// TIA Portal project "WintonWasher_Recycler" (V15)

(* hardware
DEVICE "S7300/ET200M station_1"  S7-300 station
   slot 0: "Rail_0"  Rail  6ES7 390-1***0-0AA0
   slot 2: "PLC_1"  CPU 315-2 PN/DP  6ES7 315-2EH14-0AB0  V3.2
      slot 2: "PROFINET interface_1"  PN-IO
         slot 1: "Port_1"  Port
         slot 2: "Port_2"  Port
   slot 4: "DI 32x24VDC_1"  DI32 x 24VDC  6ES7 321-1BL00-0AA0
   slot 5: "DO 32x24VDC/0.5A_1"  DO32 x 24VDC / 0.5A  6ES7 322-1BL00-0AA0
DEVICE "HMI_1"  TP700 Comfort
   slot 0: "HMI_1"  TP700 Comfort  6AV2 124-0GC01-0AX0  15.0.0.0
   slot 1: "HMI_RT_1"  TP700 Comfort  6AV2 124-0GC01-0AX0  15.0.0.0
   slot 5: "HMI_1.IE_CP_1"  PROFINET Interface  15.0.0.0
      slot 1: "PROFINET Interface_1"  PROFINET Interface
         slot 1: "Port_1"  Port
         slot 2: "Port_2"  Port
   slot 7: "HMI_1.MPI/DP_CP_1"  MPI/DP Interface  15.0.0.0
DEVICE "GSD device_1"  GSD.Device
   slot 0: "Rack_0"  Rail
*)

// ===== PLC "PLC_1"  CPU 315-2 PN/DP =====

VAR_GLOBAL   // PLC tag table "Ouput Tag Table"
   "Qx Shear Cyl Ret" AT %Q10.0 : Bool;
   "Qx Shear Cyl Ext" AT %Q10.1 : Bool;   // lateral must be ret, punch must be ret
   "Qx Prestop Cyl Ret" AT %Q10.2 : Bool;   // RET lets part through
   "Qx Prestop Cyl Ext" AT %Q10.3 : Bool;
   "Qx Endstop Cyl Ret" AT %Q10.4 : Bool;   // prestop must be ext,
   "Qx Endstop Cyl Ext" AT %Q10.5 : Bool;
   "Qx Clamp Cyl Ret" AT %Q10.6 : Bool;
   "Qx Clamp Cyl Ext" AT %Q10.7 : Bool;
   "Qx Punch Cyl Ret" AT %Q11.0 : Bool;
   "Qx Punch Cyl Ext" AT %Q11.1 : Bool;
   "Qx Gripper Cyl Ret" AT %Q12.0 : Bool;
   "Qx Gripper Cyl Ext" AT %Q12.1 : Bool;
   "Qx Lat Cyl Ret" AT %Q12.2 : Bool;
   "Qx Lat Cyl Ext" AT %Q12.3 : Bool;   // Prestop must be EXT, gripper ret, endstop must be RET, punch ret, shear ret, clamps ret
   "Qx T2 Cyl Ret" AT %Q12.4 : Bool;
   "Qx T2 Cyl Ext" AT %Q12.5 : Bool;
   "Qx T1 Cyl Ret" AT %Q12.6 : Bool;
   "Qx T1 Cyl Ext" AT %Q12.7 : Bool;
   "Qx Cycle Start PL" AT %Q5.0 : Bool;
   "Qx Feeder OFF" AT %Q5.1 : Bool;   // Logic is Reversed!
   "Qx Overhead Light ON" AT %Q5.2 : Bool;
   "Qx Fan ON" AT %Q5.3 : Bool;
   "Qx Auxiliary Lights ON" AT %Q5.4 : Bool;
END_VAR

VAR_GLOBAL   // PLC tag table "Input Tag Table"
   "Ix Prestop Ext PX" AT %I10.2 : Bool;
   "Ix Prestop Ret PX" AT %I10.3 : Bool;
   "Ix Endstop Ext PX" AT %I10.4 : Bool;
   "Ix Endstop Ret PX" AT %I10.5 : Bool;
   "Ix Punch Ext PX" AT %I10.6 : Bool;
   "Ix Punch Ret PX" AT %I10.7 : Bool;
   "Ix Washer Present PX" AT %I11.0 : Bool;
   "Ix Left Clamp Ext PX" AT %I11.2 : Bool;
   "Ix Left Clamp Ret PX" AT %I11.3 : Bool;
   "Ix Right Clamp Ext PX" AT %I11.4 : Bool;
   "Ix Right Clamp Ret PX" AT %I11.5 : Bool;
   "Ix Left Shear Ext PX" AT %I11.6 : Bool;
   "Ix Left Shear Ret PX" AT %I11.7 : Bool;
   "Backup Washer Present PX" AT %I11.1 : Bool;
   "Ix Gripper Ext PX" AT %I12.0 : Bool;
   "Ix Gripper Ret PX" AT %I12.1 : Bool;
   "Ix Lat Ext PX" AT %I12.2 : Bool;
   "Ix Lat Ret PX" AT %I12.3 : Bool;
   "Ix T2 Ext PX" AT %I12.4 : Bool;
   "Ix T2 Ret PX" AT %I12.5 : Bool;
   "Ix T1 Ext PX" AT %I12.6 : Bool;
   "Ix T1 Ret PX" AT %I12.7 : Bool;
   "Ix Sense Part Ready PE" AT %I13.4 : Bool;
   "Ix Right Shear Ext PX" AT %I13.6 : Bool;
   "Ix Right Shear Ret PX" AT %I13.7 : Bool;
   "Ix Cycle Start PB" AT %I1.0 : Bool;
   "Ix ESTOP Not Pressed" AT %I1.1 : Bool;
   "Ix Doors Are Closed" AT %I1.2 : Bool;
END_VAR

DATA_BLOCK "DB_WintonWasher"   // DB1
{ S7_Optimized_Access := 'FALSE' }
VERSION : 0.1
// stored: InstanceOfName FB_WintonWasher
"FB_WintonWasher"
BEGIN
END_DATA_BLOCK

DATA_BLOCK "HMI_DB"   // DB7
{ S7_Optimized_Access := 'FALSE' }
VERSION : 0.1
   VAR
      MasterReset : Bool;
      Pause : Bool;
      "Auto On" : Bool;
      "Punch Ext" : Bool;
      "Punch Ret" : Bool;
      "Shear Ext" : Bool;
      "Shear Ret" : Bool;
      "Prestop Ext" : Bool;
      "Prestop Ret" : Bool;
      "Endstop Ext" : Bool;
      "Endstop Ret" : Bool;
      "Clamp Ext" : Bool;
      "Clamp Ret" : Bool;
      "Gripper Ext" : Bool;
      "Gripper Ret" : Bool;
      "Lat Ext" : Bool;
      "Lat Ret" : Bool;
      "T1 Ext" : Bool;
      "T1 Ret" : Bool;
      "T2 Ext" : Bool;
      "T2 Ret" : Bool;
      Vibrate : Bool;
      "Overhead Lights" : Bool;
      "Auxiliary Lights" : Bool;
      Fan : Bool;
      Bin_Count : Int;
      Reset_Bin_Count : Bool;
      Cycle_Count : Int;
   END_VAR
BEGIN
END_DATA_BLOCK

DATA_BLOCK "Alarms_DB"   // DB11
{ S7_Optimized_Access := 'FALSE' }
VERSION : 0.1
   VAR
      Alarms : Word;
   END_VAR
BEGIN
END_DATA_BLOCK

FUNCTION_BLOCK "FB_WintonWasher"   // FB1, STL
TITLE = Winton Washer Recycler
{ S7_Optimized_Access := 'FALSE' }
VERSION : 0.1
// Winton Washer Recycler Program
   VAR_INPUT
      "ESTOP Pressed" : Bool;
      "Ix Doors are Closed" : Bool;
      "Ix Prestop Ext PX" : Bool;
      "Ix Prestop Ret PX" : Bool;
      "Ix Endstop Ext PX" : Bool;
      "Ix Endstop Ret PX" : Bool;
      "Ix Punch Ext PX" : Bool;
      "Ix Punch Ret PX" : Bool;
      "Ix Washer Present PX" : Bool;
      "Ix Left Clamp Ext PX" : Bool;
      "Ix Left Clamp Ret PX" : Bool;
      "Ix Right Clamp Ext PX" : Bool;
      "Ix Right Clamp Ret PX" : Bool;
      "Ix Left Shear Ext PX" : Bool;
      "Ix Left Shear Ret PX" : Bool;
      "Backup Washer Present PX" : Bool;
      "Ix Gripper Ext PX" : Bool;
      "Ix Gripper Ret PX" : Bool;
      "Ix Lat Ext PX" : Bool;
      "Ix Lat Ret PX" : Bool;
      "Ix T2 Ext PX" : Bool;
      "Ix T2 Ret PX" : Bool;
      "Ix T1 Ext PX" : Bool;
      "Ix T1 Ret PX" : Bool;
      "Ix Sense Part Ready PE" : Bool;
      "Ix Right Shear Ext PX" : Bool;
      "Ix Right Shear Ret PX" : Bool;
      "Ix Cycle Start PB" : Bool;
   END_VAR
   VAR_OUTPUT
      "Qx Shear Cyl Ret" : Bool;
      "Qx Shear Cyl Ext" : Bool;
      "Qx Prestop Cyl Ret" : Bool;
      "Qx Prestop Cyl Ext" : Bool;
      "Qx Endstop Cyl Ret" : Bool;
      "Qx Endstop Cyl Ext" : Bool;
      "Qx Clamp Cyl Ret" : Bool;
      "Qx Clamp Cyl Ext" : Bool;
      "Qx Punch Cyl Ret" : Bool;
      "Qx Punch Cyl Ext" : Bool;
      "Qx Gripper Cyl Ret" : Bool;
      "Qx Gripper Cyl Ext" : Bool;
      "Qx Lat Cyl Ret" : Bool;
      "Qx Lat Cyl Ext" : Bool;
      "Qx T2 Cyl Ret" : Bool;
      "Qx T2 Cyl Ext" : Bool;
      "Qx T1 Cyl Ret" : Bool;
      "Qx T1 Cyl Ext" : Bool;
      "Qx Cycle Start PL" : Bool;
      "Qx Feeder OFF" : Bool;
      "Qx Overhead Light ON" : Bool;
      "Qx Fan ON" : Bool;
      "Qx Auxiliary Lights ON" : Bool;
   END_VAR
   VAR
      "Master Reset" : Bool;
      Pause : Bool;
      Auto : Struct
         "Shear Cyl Ret" : Bool;
         "Shear Cyl Ext" : Bool;
         "Prestop Cyl Ret" : Bool;
         "Prestop Cyl Ext" : Bool;
         "Endstop Cyl Ret" : Bool;
         "Endstop Cyl Ext" : Bool;
         "Clamp Cyl Ret" : Bool;
         "Clamp Cyl Ext" : Bool;
         "Punch Cyl Ret" : Bool;
         "Punch Cyl Ext" : Bool;
         "Gripper Cyl Ret" : Bool;
         "Gripper Cyl Ext" : Bool;
         "Lat Cyl Ret" : Bool;
         "Lat Cyl Ext" : Bool;
         "T2 Cyl Ret" : Bool;
         "T2 Cyl Ext" : Bool;
         "T1 Cyl Ret" : Bool;
         "T1 Cyl Ext" : Bool;
         "Cycle Start PL" : Bool;
         "Feeder OFF" : Bool;
      END_STRUCT;
      Manual : Struct
         "Shear Cyl Ret" : Bool;
         "Shear Cyl Ext" : Bool;
         "Prestop Cyl Ret" : Bool;
         "Prestop Cyl Ext" : Bool;
         "Endstop Cyl Ret" : Bool;
         "Endstop Cyl Ext" : Bool;
         "Clamp Cyl Ret" : Bool;
         "Clamp Cyl Ext" : Bool;
         "Punch Cyl Ret" : Bool;
         "Punch Cyl Ext" : Bool;
         "Gripper Cyl Ret" : Bool;
         "Gripper Cyl Ext" : Bool;
         "Lat Cyl Ret" : Bool;
         "Lat Cyl Ext" : Bool;
         "T2 Cyl Ret" : Bool;
         "T2 Cyl Ext" : Bool;
         "T1 Cyl Ret" : Bool;
         "T1 Cyl Ext" : Bool;
         "Cycle Start PL" : Bool;
         "Feeder OFF" : Bool;
         "Light ON" : Bool;
         "Fan ON" : Bool;
      END_STRUCT;
      "Step" : Struct
         Idle : Bool;
         "Sense Part Ready" : Bool;
         "Activate Prestop" : Bool;
         "Pick and Place Retract Endstop" : Bool;
         "Pick and Place Extend Lat Cyl" : Bool;
         "Pick and Place Extend Clamp" : Bool;
         "Pick and Place Extend Gripper" : Bool;
         "Pick and Place Retract Lat Cyl" : Bool;
         "Pick and Place Retract Gripper" : Bool;
         "Pick and Place Extend Endstop" : Bool;
         "Check for Washer" : Bool;
         "Open Path to Head Bin" : Bool;
         "Remove Head" : Bool;
         "Open Path to  Washer Bin" : Bool;
         "Retract Shears" : Bool;
         "Punch Out Washer" : Bool;
         "Retract Punch" : Bool;
         "Open Path to Body Bin" : Bool;
         "Drop Part" : Bool;
      END_STRUCT;
      Transition1_OK : Bool;
      Transition2_OK : Bool;
      Okay_toDelay1 : Bool;
      No_Parts_Error : Bool;
      "Enable PL Blink" : Bool;
      "Enable Overhead Blink" : Bool;
      Start_Delay_OffVibrate : Bool;
      Stop_Vibrate : Bool;   // timer output variable to stop feeder
      Washer_NotPresent : Bool;
      Bin_Overflow : Bool;
      Cyl_Jam : Bool;
      ClearPart : Struct
         "Retract Shears" : Bool;
         "Retract Punch" : Bool;
         "Extend Gripper" : Bool;
         "Retract Endstop" : Bool;
         "Extend Prestop" : Bool;
         "Retract Lateral" : Bool;
         "Retract Clamp" : Bool;
         "Reset Cyls for Idle" : Bool;
      END_STRUCT;
      "Start _Timeout" : Bool;
      Start_PreExt_Jam : Bool;
      Start_PreRet_Jam : Bool;
      Start_EndExt_Jam : Bool;
      Start_EndRet_Jam : Bool;
      Start_GrpExt_Jam : Bool;
      Start_GrpRet_Jam : Bool;
      Start_LatExt_Jam : Bool;
      Start_LatRet_Jam : Bool;
      Start_ShrExt_Jam : Bool;
      Start_ShrRet_Jam : Bool;
      Start_PunExt_Jam : Bool;
      Start_PunRet_Jam : Bool;
      Start_T1Ext_Jam : Bool;
      Start_T1Ret_Jam : Bool;
      Start_T2Ext_Jam : Bool;
      Start_T2Ret_Jam : Bool;
      Start_ClmpExt_Jam : Bool;
      Start_ClmpRet_Jam : Bool;
   END_VAR
BEGIN

REGION Network 1: Reset and Pause
   // Reset Conditions
   // Resets current machine state to Idle
   // HMI 'MASTER RESET' for cylinder fault or jam. 
   // -This button will automatically clear a part and reset cylinder positions to where they should be in Idle.
   ////////////////////////////////////////////////////
   //--------------Master Reset Conditions-------------
         A     #"ESTOP Pressed";
         =     #"Master Reset";

   ////////////////////////////////////////////////////
   //--------------Reset State Condition-------------
   //add other errors
         A     #"Master Reset";
         O     #No_Parts_Error;
         O(;
   //logic from "Clear part" sequence
         A     #ClearPart."Reset Cyls for Idle";
         A     #"Ix Gripper Ret PX";
         A     #"Ix Endstop Ext PX";
         A     #"Ix T1 Ret PX";
         A     #"Ix T2 Ext PX";
         );
         S     #"Step".Idle;
         R     #"Step"."Activate Prestop";
         R     #"Step"."Check for Washer";
         R     #"Step"."Drop Part";
         R     #"Step"."Open Path to  Washer Bin";
         R     #"Step"."Open Path to Body Bin";
         R     #"Step"."Open Path to Head Bin";
         R     #"Step"."Pick and Place Retract Endstop";
         R     #"Step"."Pick and Place Extend Lat Cyl";
         R     #"Step"."Pick and Place Extend Clamp";
         R     #"Step"."Pick and Place Extend Gripper";
         R     #"Step"."Pick and Place Retract Lat Cyl";
         R     #"Step"."Pick and Place Retract Gripper";
         R     #"Step"."Pick and Place Extend Endstop";
         R     #"Step"."Punch Out Washer";
         R     #"Step"."Remove Head";
         R     #"Step"."Retract Shears";
         R     #"Step"."Sense Part Ready";
         R     #ClearPart."Extend Gripper";
         R     #ClearPart."Extend Prestop";
         R     #ClearPart."Reset Cyls for Idle";
         R     #ClearPart."Retract Clamp";
         R     #ClearPart."Retract Endstop";
         R     #ClearPart."Retract Lateral";
         R     #ClearPart."Retract Punch";
         R     #ClearPart."Retract Shears";



   //////////////////////////////////////////////////////
   //--------------HMI Master Reset Response-------------
   //start clear part sequence
         A     "HMI_DB".MasterReset;
         S     #ClearPart."Retract Shears";
         R     #"Step"."Activate Prestop";
         R     #"Step"."Check for Washer";
         R     #"Step"."Drop Part";
         R     #"Step"."Open Path to  Washer Bin";
         R     #"Step"."Open Path to Body Bin";
         R     #"Step"."Open Path to Head Bin";
         R     #"Step"."Pick and Place Retract Endstop";
         R     #"Step"."Pick and Place Extend Lat Cyl";
         R     #"Step"."Pick and Place Extend Clamp";
         R     #"Step"."Pick and Place Extend Gripper";
         R     #"Step"."Pick and Place Retract Lat Cyl";
         R     #"Step"."Pick and Place Retract Gripper";
         R     #"Step"."Pick and Place Extend Endstop";
         R     #"Step"."Punch Out Washer";
         R     #"Step"."Remove Head";
         R     #"Step"."Retract Shears";
         R     #"Step"."Sense Part Ready";
         R     #"Step".Idle;

   ////////////////////////////////////////////
   //--------------Pause Logic-----------------
         AN    #"Ix Doors are Closed";
   // ON    "HMI_DB"."Auto On"
         O     "HMI_DB".Pause;
         =     #Pause;

   //use this timer to generate any delay desired
   //CALL  TON , "CylJam_Timer"
   //         time_type:=Time
   //         IN :=#Step."Retract Shears"
   //         PT :=T#2s
   //         Q  :=#Auto."Shear Cyl Ret"
   //         ET :=
END_REGION

REGION Network 2: Manual Network
   // Manual Control of all Outputs via HMI
   ////////////////////////////////////////////
   //--------------Manual: Prestop-------------
         A     "HMI_DB"."Prestop Ext";
         AN    "HMI_DB"."Auto On";
         =     #Manual."Prestop Cyl Ext";

         A     "HMI_DB"."Prestop Ret";
         AN    "HMI_DB"."Auto On";
         =     #Manual."Prestop Cyl Ret";

   ////////////////////////////////////////////
   //--------------Manual: Endsotp-------------
         A     "HMI_DB"."Endstop Ext";
         AN    "HMI_DB"."Auto On";
         =     #Manual."Endstop Cyl Ext";

         A     "HMI_DB"."Endstop Ret";
         AN    "HMI_DB"."Auto On";
         =     #Manual."Endstop Cyl Ret";

   ////////////////////////////////////////////
   //--------------Manual: Lateral-------------
         A     "HMI_DB"."Lat Ext";
         AN    "HMI_DB"."Auto On";
         =     #Manual."Lat Cyl Ext";

         A     "HMI_DB"."Lat Ret";
         AN    "HMI_DB"."Auto On";
         =     #Manual."Lat Cyl Ret";

   ////////////////////////////////////////////
   //--------------Manual: Gripper-------------
         A     "HMI_DB"."Gripper Ext";
         AN    "HMI_DB"."Auto On";
         =     #Manual."Gripper Cyl Ext";

         A     "HMI_DB"."Gripper Ret";
         AN    "HMI_DB"."Auto On";
         =     #Manual."Gripper Cyl Ret";

   ////////////////////////////////////////////
   //--------------Manual: Shears-------------
         A     "HMI_DB"."Shear Ext";
         AN    "HMI_DB"."Auto On";
         =     #Manual."Shear Cyl Ext";

         A     "HMI_DB"."Shear Ret";
         AN    "HMI_DB"."Auto On";
         =     #Manual."Shear Cyl Ret";

   ////////////////////////////////////////////
   //--------------Manual: Clamps-------------
         A     "HMI_DB"."Clamp Ext";
         AN    "HMI_DB"."Auto On";
         =     #Manual."Clamp Cyl Ext";

         A     "HMI_DB"."Clamp Ret";
         AN    "HMI_DB"."Auto On";
         =     #Manual."Clamp Cyl Ret";

   ////////////////////////////////////////////
   //--------------Manual: Washer Punch-------------
         A     "HMI_DB"."Punch Ext";
         AN    "HMI_DB"."Auto On";
         =     #Manual."Punch Cyl Ext";

         A     "HMI_DB"."Punch Ret";
         AN    "HMI_DB"."Auto On";
         =     #Manual."Punch Cyl Ret";

   ////////////////////////////////////////////
   //--------------Manual: Trap Door 1-------------
         A     "HMI_DB"."T1 Ext";
         AN    "HMI_DB"."Auto On";
         =     #Manual."T1 Cyl Ext";

         A     "HMI_DB"."T1 Ret";
         AN    "HMI_DB"."Auto On";
         =     #Manual."T1 Cyl Ret";


   ////////////////////////////////////////////
   //--------------Manual: Trap Door 2-------------
         A     "HMI_DB"."T2 Ext";
         AN    "HMI_DB"."Auto On";
         =     #Manual."T2 Cyl Ext";

         A     "HMI_DB"."T2 Ret";
         AN    "HMI_DB"."Auto On";
         =     #Manual."T2 Cyl Ret";

   ////////////////////////////////////////////
   //--------------Manual: Vibrate Feeder-------------
         AN    "HMI_DB".Vibrate;
         AN    "HMI_DB"."Auto On";
         =     #Manual."Feeder OFF";
END_REGION

REGION Network 3: Auto Sequence - Step Transitions
   // How the auto sequence transitions states
   ////////////////////////////////////////////////////
   //-------------Idle to Sense Part Ready-------------
         A     #"Step".Idle;
         R     #ClearPart."Reset Cyls for Idle";

         A     #"Step".Idle;
         A     #"Ix Cycle Start PB";
         A     "HMI_DB"."Auto On";
         AN    #Pause;
         AN    "Bin_Count".Q;
         R     #"Step".Idle;
         S     #"Step"."Sense Part Ready";


   ////////////////////////////////////////////////////
   //--------sense part ready to activate prestop------
         A     #"Step"."Sense Part Ready";
         A     #"Ix Sense Part Ready PE";
         A     "HMI_DB"."Auto On";
         AN    #Pause;
         S     #"Step"."Activate Prestop";
         R     #"Step"."Sense Part Ready";

         A     #"Step"."Sense Part Ready";
         AN    "Bin_Count".Q;
         =     #"Start _Timeout";

   //No parts timeout delay
         CALL  TON , "No Parts Timeout Timer"
         ( IN := #"Start _Timeout",
           PT := T#30s,
           Q  := #No_Parts_Error,
           ET :=
         );

   ////////////////////////////////////////////////////
   //-------Activate prestop to Pick and Place---------
         A     #"Step"."Activate Prestop";
         A     #"Ix Prestop Ext PX";
         A     "HMI_DB"."Auto On";
         AN    #Pause;
         S     #"Step"."Pick and Place Retract Endstop";
         R     #"Step"."Activate Prestop";

   ////////////////////////////////////////////////////
   //---------------Pick and place---------------------
   //---------------retract endstop--------------------
         A     #"Step"."Pick and Place Retract Endstop";
         A     #"Ix Endstop Ret PX";
         A     "HMI_DB"."Auto On";
         AN    #Pause;
         R     #"Step"."Pick and Place Retract Endstop";
         S     #"Step"."Pick and Place Extend Lat Cyl";

   ////////////////////////////////////////////////////
   //---------------Pick and place---------------------
   //---------------Extend Lateral---------------------
         A     #"Step"."Pick and Place Extend Lat Cyl";
         A     #"Ix Lat Ext PX";
         A     "HMI_DB"."Auto On";
         AN    #Pause;
         R     #"Step"."Pick and Place Extend Lat Cyl";
         S     #"Step"."Pick and Place Extend Clamp";

   ////////////////////////////////////////////////////
   //---------------Pick and place---------------------
   //---------------Extend Clamp-----------------------
         A     #"Step"."Pick and Place Extend Clamp";
         A     #"Ix Left Clamp Ext PX";
         A     #"Ix Right Clamp Ext PX";
         A     "HMI_DB"."Auto On";
         AN    #Pause;
         R     #"Step"."Pick and Place Extend Clamp";
         S     #"Step"."Pick and Place Extend Gripper";

   ////////////////////////////////////////////////////
   //---------------Pick and place---------------------
   //---------------Extend Gripper---------------------
         A     #"Step"."Pick and Place Extend Gripper";
         A     #"Ix Gripper Ext PX";
         A     "HMI_DB"."Auto On";
         AN    #Pause;
         R     #"Step"."Pick and Place Extend Gripper";
         S     #"Step"."Pick and Place Retract Lat Cyl";

   ////////////////////////////////////////////////////
   //---------------Pick and place---------------------
   //---------------Retract Lateral--------------------
         A     #"Step"."Pick and Place Retract Lat Cyl";
         A     #"Ix Lat Ret PX";
         A     "HMI_DB"."Auto On";
         AN    #Pause;
         R     #"Step"."Pick and Place Retract Lat Cyl";
         S     #"Step"."Pick and Place Retract Gripper";

   ////////////////////////////////////////////////////
   //---------------Pick and place---------------------
   //---------------Retract Gripper--------------------
         A     #"Step"."Pick and Place Retract Gripper";
         A     #"Ix Gripper Ret PX";
         A     "HMI_DB"."Auto On";
         AN    #Pause;
         R     #"Step"."Pick and Place Retract Gripper";
         S     #"Step"."Pick and Place Extend Endstop";

   ////////////////////////////////////////////////////
   //---------------Pick and place---------------------
   //---------------Extend Endstop--------------------
         A     #"Step"."Pick and Place Extend Endstop";
         A     #"Ix Endstop Ext PX";
         A     "HMI_DB"."Auto On";
         AN    #Pause;
         R     #"Step"."Pick and Place Extend Endstop";
         S     #"Step"."Check for Washer";

   ////////////////////////////////////////////////////
   //----check for washer to Open Path to Head Bin-----
         A     #"Step"."Check for Washer";
         A     #"Ix Washer Present PX";
         A     "HMI_DB"."Auto On";
         AN    #Pause;
         R     #"Step"."Check for Washer";
         S     #"Step"."Open Path to Head Bin";

   //else
   //timer, put output of timer on Drop part conditions

   ////////////////////////////////////////////////////
   //---------check for washer to Drop part, put in condition for drp part
         CALL  TON , "Washer Not Present Timeout Timer"
         ( IN := #"Step"."Check for Washer",
           PT := T#100ms,
           Q  := #Washer_NotPresent,
           ET :=
         );

   //      A     #Step."Check for Washer"
   //      A   Check for Washer Timeout
   //      S     #Step."Drop Part"
   //      R     #Step."Check for Washer"

   ////////////////////////////////////////////////////
   //---------Open Path to Head Bin, to Remove Head---
         A     #"Step"."Open Path to Head Bin";
         A     #"Ix T1 Ext PX";
         A     #"Ix T2 Ext PX";
         A     "HMI_DB"."Auto On";
         AN    #Pause;
         S     #"Step"."Remove Head";
         R     #"Step"."Open Path to Head Bin";

   ////////////////////////////////////////////////////
   //------Remove Head, to Open Path to Washer Bin-----
   //start delay after Extension
         A     #"Step"."Remove Head";
         A     #"Ix Left Shear Ext PX";
         =     #Okay_toDelay1;

   //delay
         CALL  TON , "Delay_Transition_toWasherBin"
         ( IN := #Okay_toDelay1,
           PT := T#1s,
           Q  := #Transition1_OK,
           ET :=
         );

         A     #"Step"."Remove Head";
         A     #"Ix Left Shear Ext PX";
         A     #"Ix Right Shear Ext PX";
         A     #Transition1_OK;
         A     "HMI_DB"."Auto On";
         AN    #Pause;
         R     #"Step"."Remove Head";
         S     #"Step"."Open Path to  Washer Bin";

   ////////////////////////////////////////////////////
   //-----Open Path to Washer Bin to Retract Shears----
         A     #"Step"."Open Path to  Washer Bin";
         A     #"Ix T1 Ext PX";
         A     #"Ix T2 Ret PX";
         A     "HMI_DB"."Auto On";
         AN    #Pause;
         R     #"Step"."Open Path to  Washer Bin";
         S     #"Step"."Retract Shears";

   ////////////////////////////////////////////////////
   //---------Retract Shears to Punch Out Washer-------
         A     #"Step"."Retract Shears";
         A     #"Ix Left Shear Ret PX";
         A     #"Ix Right Shear Ret PX";
         A     "HMI_DB"."Auto On";
         AN    #Pause;
         R     #"Step"."Retract Shears";
         S     #"Step"."Punch Out Washer";


   ////////////////////////////////////////////////////
   //-----Punch Out Washer to Retract Punch----
         A     #"Step"."Punch Out Washer";
         A     #"Ix Punch Ext PX";
         A     "HMI_DB"."Auto On";
         AN    #Pause;
         R     #"Step"."Punch Out Washer";
         S     #"Step"."Retract Punch";

   ////////////////////////////////////////////////////
   //-----Retract Punch to Open Path to Body Bin-------
   //delay
         CALL  TON , "Delay_Transition_toBodyBin"
         ( IN := #"Step"."Retract Punch",
           PT := T#1s,
           Q  := #Transition2_OK,
           ET :=
         );

         A     #"Step"."Retract Punch";
         A     #"Ix Punch Ret PX";
         A     "HMI_DB"."Auto On";
         AN    #Pause;
         A     #Transition2_OK;
         R     #"Step"."Retract Punch";
         S     #"Step"."Open Path to Body Bin";

   ////////////////////////////////////////////////////
   //-------Open Pach to Body Bin to Drop Part---------
         A(;
         A     #"Step"."Open Path to Body Bin";
         A     #"Ix T1 Ret PX";
         );
         O(;
         A     #"Step"."Check for Washer";
         A     #Washer_NotPresent;
         );
         A     "HMI_DB"."Auto On";
         AN    #Pause;
         R     #"Step"."Open Path to Body Bin";
         R     #"Step"."Check for Washer";
         S     #"Step"."Drop Part";

   ////////////////////////////////////////////////////
   //---------Drop Part to Wait for Part Ready---------
         A     #"Step"."Drop Part";
         A     #"Ix Left Clamp Ret PX";
         A     #"Ix Right Clamp Ret PX";
         A     "HMI_DB"."Auto On";
         AN    #Pause;
         R     #"Step"."Drop Part";
         S     #"Step"."Sense Part Ready";
END_REGION

REGION Network 4: Auto Sequence - Outputs
   ////////////////////////////////////////////////////////////////////////
   //--------------------------Idle----------------------------------------

   //cycle start PL
         A     #"Step".Idle;
         A     "HMI_DB"."Auto On";
         AN    "PL_Blink".Q;
         =     #"Enable PL Blink";

         CALL  TON , "PL_Blink"
         ( IN := #"Enable PL Blink",
           PT := T#1s,
           Q  := ,
           ET :=
         );


         AN    #"Step".Idle;
         AN    #Pause;
         A     "HMI_DB"."Auto On";
         AN    "HMI_DB".MasterReset;
         O(;
         L     "PL_Blink".ET;
         L     T#500ms;
         >D;
         );
         =     #Auto."Cycle Start PL";

   ////////////////////////////////////////////////////////////////////////
   //--------------------------Sense Part Ready----------------------------
   //     A     #"Ix Sense Part Ready PE"
   //   AN    "Bin_Count".Q
   //  =     #Start_Delay_OffVibrate

   //Vibrating Feeder control (inversed)
   //delay after seeing part to remove time inbetween cycles
         CALL  TOF , "Delay_VibrateOFF"
         ( IN := #"Ix Sense Part Ready PE",
           PT := T#2s,
           Q  := #Stop_Vibrate,
           ET :=
         );

   //if neither are true, it is OFF
         AN    #"Step"."Sense Part Ready";
         AN    #Stop_Vibrate;
         ON    "HMI_DB"."Auto On";
         O     #"Master Reset";
         O     "Bin_Count".Q;
         =     #Auto."Feeder OFF";

   //retract prestop
         A     #"Step"."Sense Part Ready";
         =     #Auto."Prestop Cyl Ret";

   ////////////////////////////////////////////////////////////////////////
   //--------------------------Activate Prestop----------------------------
   //Extend Prestop
         A     #"Step"."Activate Prestop";
         =     #Auto."Prestop Cyl Ext";

   ////////////////////////////////////////////////////////////////////////
   //-----------------Pick and Place Retract Endstop-----------------------
   //retract endstop
         A     #"Step"."Pick and Place Retract Endstop";
         =     #Auto."Endstop Cyl Ret";

   ////////////////////////////////////////////////////////////////////////
   //-----------------Pick and Place Extend Lat Cyl-----------------------
   //retract endstop
         A     #"Step"."Pick and Place Extend Lat Cyl";
         =     #Auto."Lat Cyl Ext";

   ////////////////////////////////////////////////////////////////////////
   //-----------------Pick and Place Extend Clamp-----------------------
         A     #"Step"."Pick and Place Extend Clamp";
         =     #Auto."Clamp Cyl Ext";

   ////////////////////////////////////////////////////////////////////////
   //-----------------Pick and Place Extend Gripper-----------------------
         A     #"Step"."Pick and Place Extend Gripper";
         =     #Auto."Gripper Cyl Ext";

   ////////////////////////////////////////////////////////////////////////
   //-----------------Pick and Place Retract Lateral-----------------------
         A     #"Step"."Pick and Place Retract Lat Cyl";
         =     #Auto."Lat Cyl Ret";

   ////////////////////////////////////////////////////////////////////////
   //-----------------Pick and Place Retract Gripper-----------------------
         A     #"Step"."Pick and Place Retract Gripper";
         =     #Auto."Gripper Cyl Ret";

   ////////////////////////////////////////////////////////////////////////
   //-----------------Pick and Place Extend Endstop-----------------------
         A     #"Step"."Pick and Place Extend Endstop";
         =     #Auto."Endstop Cyl Ext";

   ////////////////////////////////////////////////////////////////////////
   //-------------------------Check for Washer-----------------------------

   ////////////////////////////////////////////////////////////////////////
   //-----------------------Open Path(s) logic--------------------------

   //T1
         A     #"Step"."Open Path to Head Bin";
         O     #"Step"."Open Path to  Washer Bin";
         =     #Auto."T1 Cyl Ext";

   //T2
         A     #"Step"."Open Path to Head Bin";
         O     #"Step"."Open Path to Body Bin";
         =     #Auto."T2 Cyl Ext";


   //T1
         A     #"Step"."Open Path to Body Bin";
         =     #Auto."T1 Cyl Ret";

   //T2
         A     #"Step"."Open Path to  Washer Bin";
         =     #Auto."T2 Cyl Ret";

   ////////////////////////////////////////////////////////////////////////
   //---------------------------Remove Head--------------------------------
         A     #"Step"."Remove Head";
         =     #Auto."Shear Cyl Ext";

   ////////////////////////////////////////////////////////////////////////
   //-------------------------Open Path to Washer Bin-----------------------------
   //this logic is with the T1 and T2 logic

   ////////////////////////////////////////////////////////////////////////
   //-------------------------Retract Shears-----------------------------
         A     #"Step"."Retract Shears";
         =     #Auto."Shear Cyl Ret";

   ////////////////////////////////////////////////////////////////////////
   //-------------------------Punch Out Washer-----------------------------
         A     #"Step"."Punch Out Washer";
         =     #Auto."Punch Cyl Ext";

   ////////////////////////////////////////////////////////////////////////
   //-------------------------Retract Punch-----------------------------
         A     #"Step"."Retract Punch";
         =     #Auto."Punch Cyl Ret";


   ////////////////////////////////////////////////////////////////////////
   //-------------------------Drop Part-----------------------------
         A     #"Step"."Drop Part";
         =     #Auto."Clamp Cyl Ret";

         CALL  CTU, "Bin_Count"
         ( CU := #"Step"."Drop Part",
           R  := "HMI_DB".Reset_Bin_Count,
           PV := 135,
           Q  := #Bin_Overflow,
           CV := "HMI_DB".Bin_Count
         );

         CALL  CTU , "Cycle_Count"
         ( CU := #"Step"."Drop Part",
           R  := ,
           PV := 32767,
           Q  := ,
           CV := "HMI_DB".Cycle_Count
         );


   //and increment a monthly cycle count
END_REGION

REGION Network 5: Outputs
   // Output Buffering
   ////////////////////////////////////////////////////////////////////////
   //-----------------------PLC Output Card--------------------------------

   //feeder
         A     #Auto."Feeder OFF";
         O(;
         A     #"Step".Idle;
         A     #Manual."Feeder OFF";
         AN    "HMI_DB"."Auto On";
         );
         O     #Cyl_Jam;
         O     #"Master Reset";
         =     #"Qx Feeder OFF";

   //overhead light, manually controlled
         A     "HMI_DB"."Overhead Lights";
         AN    #Cyl_Jam;
         O(;
         L     "Overhead_Blink".ET;
         L     T#500ms;
         >D;
         );
         =     #"Qx Overhead Light ON";

   //Aux Lights, manually controlled
         A     "HMI_DB"."Auxiliary Lights";
         =     #"Qx Auxiliary Lights ON";

   //Fan, manually controlled
         A     "HMI_DB".Fan;
         =     #"Qx Fan ON";

   //cycle start pilot light
         A     #Auto."Cycle Start PL";
         =     #"Qx Cycle Start PL";

   ////////////////////////////////////////////////////////////////////////
   //-----------------------Output Bank Cyls--------------------------------
   //////////////-----Contains interlocking cyl conditions-------///////////
   ////prestop
         A     #Auto."Prestop Cyl Ext";
         O     #ClearPart."Extend Prestop";
         O     #Manual."Prestop Cyl Ext";
         AN    #"Ix Prestop Ext PX";
         AN    #Cyl_Jam;
         =     #"Qx Prestop Cyl Ext";

         A     #Auto."Prestop Cyl Ret";
         O     #Manual."Prestop Cyl Ret";
         AN    #"Ix Prestop Ret PX";
         AN    #Cyl_Jam;
         =     #"Qx Prestop Cyl Ret";

   ////endstop
         A     #Auto."Endstop Cyl Ext";
         O     #ClearPart."Reset Cyls for Idle";
         O     #Manual."Endstop Cyl Ext";
         AN    #"Ix Endstop Ext PX";
         AN    #Cyl_Jam;
         =     #"Qx Endstop Cyl Ext";

         A     #Auto."Endstop Cyl Ret";
         O     #ClearPart."Retract Endstop";
         O     #Manual."Endstop Cyl Ret";
         AN    #"Ix Endstop Ret PX";
         AN    #Cyl_Jam;
         =     #"Qx Endstop Cyl Ret";

   ////gripper
         A     #Auto."Gripper Cyl Ext";
         O     #ClearPart."Extend Gripper";
         O     #Manual."Gripper Cyl Ext";
         AN    #"Ix Gripper Ext PX";
         AN    #Cyl_Jam;
         =     #"Qx Gripper Cyl Ext";

         A     #Auto."Gripper Cyl Ret";
         O     #ClearPart."Reset Cyls for Idle";
         O     #Manual."Gripper Cyl Ret";
         AN    #"Ix Gripper Ret PX";
         AN    #Cyl_Jam;
         =     #"Qx Gripper Cyl Ret";

   ////lateral cyl
         A     #Auto."Lat Cyl Ext";
         O     #Manual."Lat Cyl Ext";
         A     #"Ix Prestop Ext PX";
         A     #"Ix Endstop Ret PX";
         A     #"Ix Punch Ret PX";
         A     #"Ix Left Shear Ret PX";
         A     #"Ix Right Shear Ret PX";
         A     #"Ix Left Clamp Ret PX";
         A     #"Ix Right Clamp Ret PX";
         AN    #"Ix Lat Ext PX";
         AN    #Cyl_Jam;
         =     #"Qx Lat Cyl Ext";

         A     #Auto."Lat Cyl Ret";
         O     #ClearPart."Retract Lateral";
         O     #Manual."Lat Cyl Ret";
         A     #"Ix Prestop Ext PX";
         A     #"Ix Endstop Ret PX";
         A     #"Ix Punch Ret PX";
         A     #"Ix Left Shear Ret PX";
         A     #"Ix Right Shear Ret PX";
         AN    #"Ix Lat Ret PX";
         AN    #Cyl_Jam;
         =     #"Qx Lat Cyl Ret";

   //clamp cyl
         A     #Auto."Clamp Cyl Ret";
         O     #ClearPart."Retract Clamp";
         O     #Manual."Clamp Cyl Ret";
         A(;
         ON    #"Ix Left Clamp Ret PX";
         ON    #"Ix Right Clamp Ret PX";
         );
         AN    #Cyl_Jam;
         =     #"Qx Clamp Cyl Ret";

         A(;
         A     #Auto."Clamp Cyl Ext";
         O     #Manual."Clamp Cyl Ext";
         A(;
         ON    #"Ix Left Clamp Ext PX";
         ON    #"Ix Right Clamp Ext PX";
         );
         );
   //these ensure part is clamped while sheared and punched
         O     #"Step"."Remove Head";
         AN    #Okay_toDelay1;
         O     #"Step"."Punch Out Washer";
         AN    #Cyl_Jam;
         =     #"Qx Clamp Cyl Ext";

   //T1 Cyl
         A     #Auto."T1 Cyl Ext";
         O     #Manual."T1 Cyl Ext";
         AN    #"Ix T1 Ext PX";
         AN    #Cyl_Jam;
         =     #"Qx T1 Cyl Ext";

         A     #Auto."T1 Cyl Ret";
         O     #ClearPart."Retract Shears";
         O     #Manual."T1 Cyl Ret";
         AN    #"Ix T1 Ret PX";
         AN    #Cyl_Jam;
         =     #"Qx T1 Cyl Ret";

   //T2 cyl
         A     #Auto."T2 Cyl Ext";
         O     #Manual."T2 Cyl Ext";
         O     #ClearPart."Reset Cyls for Idle";
         AN    #"Ix T2 Ext PX";
         AN    #Cyl_Jam;
         =     #"Qx T2 Cyl Ext";

         A     #Auto."T2 Cyl Ret";
         O     #Manual."T2 Cyl Ret";
         AN    #"Ix T2 Ret PX";
         AN    #Cyl_Jam;
         =     #"Qx T2 Cyl Ret";

   //shear cyl
         A     #Auto."Shear Cyl Ext";
         O     #Manual."Shear Cyl Ext";
         A     #"Ix Lat Ret PX";
         A     #"Ix Punch Ret PX";
         A(;
         ON    #"Ix Left Shear Ext PX";
         ON    #"Ix Right Shear Ext PX";
         );
         AN    #Cyl_Jam;
         =     #"Qx Shear Cyl Ext";

         A     #Auto."Shear Cyl Ret";
         O     #ClearPart."Retract Shears";
         O     #Manual."Shear Cyl Ret";
         A(;
         ON    #"Ix Left Shear Ret PX";
         ON    #"Ix Right Shear Ret PX";
         );
         AN    #Cyl_Jam;
         =     #"Qx Shear Cyl Ret";

   //punch cyl
         A     #Auto."Punch Cyl Ext";
         O     #Manual."Punch Cyl Ext";
         A     #"Ix Left Shear Ret PX";
         A     #"Ix Right Shear Ret PX";
         AN    #"Ix Punch Ext PX";
         AN    #Cyl_Jam;
         =     #"Qx Punch Cyl Ext";

         A     #Auto."Punch Cyl Ret";
         O     #ClearPart."Retract Punch";
         O     #Manual."Punch Cyl Ret";
         A     #"Ix Left Shear Ret PX";
         A     #"Ix Right Shear Ret PX";
         AN    #"Ix Punch Ret PX";
         AN    #Cyl_Jam;
         =     #"Qx Punch Cyl Ret";
END_REGION

REGION Network 6: Clear Part
   // Clears Part or Jam (potentially) from loading process. 
   // Pressing "MASTER RESET" on HMI triggers this sequence. 
   // Goes to idle when complete
   //state logic
   ////////////////////////////////////////////////////
   //---------Retract Shears to Retract Punch-------
         A     #ClearPart."Retract Shears";
         A     #"Ix Left Shear Ret PX";
         A     #"Ix Right Shear Ret PX";
         A     #"Ix T1 Ret PX";
         AN    #Pause;
         R     #ClearPart."Retract Shears";
         S     #ClearPart."Retract Punch";

   ////////////////////////////////////////////////////
   //---------Retract Punch to Extend Gripper-------
         A     #ClearPart."Retract Punch";
         A     #"Ix Punch Ret PX";
         AN    #Pause;
         R     #ClearPart."Retract Punch";
         S     #ClearPart."Extend Gripper";

   ////////////////////////////////////////////////////
   //---------Extend Gripper to Retract Endstop-------
         A(;
         A     #ClearPart."Extend Gripper";
         A     #"Ix Gripper Ext PX";
         );
         O(;
         A     #ClearPart."Extend Gripper";
         A     #"Ix Lat Ret PX";
         );
         AN    #Pause;
         R     #ClearPart."Extend Gripper";
         S     #ClearPart."Retract Endstop";

   ////////////////////////////////////////////////////
   //---------Retract Endstop to Extend Prestop-------
         A(;
         A     #ClearPart."Retract Endstop";
         A     #"Ix Endstop Ret PX";
         );
         O(;
         A     #ClearPart."Retract Endstop";
         A     #"Ix Lat Ret PX";
         );
         AN    #Pause;
         R     #ClearPart."Retract Endstop";
         S     #ClearPart."Extend Prestop";

   ////////////////////////////////////////////////////
   //---------Extend Prestop to Retract Lateral-------
         A     #ClearPart."Extend Prestop";
         A     #"Ix Prestop Ext PX";
         AN    #Pause;
         R     #ClearPart."Extend Prestop";
         S     #ClearPart."Retract Lateral";

   ////////////////////////////////////////////////////
   //---------Retract Lateral to Retract Clamp-------
         A     #ClearPart."Retract Lateral";
         A     #"Ix Lat Ret PX";
         AN    #Pause;
         R     #ClearPart."Retract Lateral";
         S     #ClearPart."Retract Clamp";

   ////////////////////////////////////////////////////
   //---------Retract Clamp to Reset Cyls For Idle-------
         A     #ClearPart."Retract Clamp";
         A     #"Ix Left Clamp Ret PX";
         A     #"Ix Right Clamp Ret PX";
         AN    #Pause;
         R     #ClearPart."Retract Clamp";
         S     #ClearPart."Reset Cyls for Idle";

   ///////////////////////////////////////////////
   //reset other cyls
   //this logic is actually in "Idle" logic because it must be in the same 'rung'
   //   A     #ClearPart."Reset Cyls for Idle"
   //   A     #"Ix Gripper Ret PX"
   //   A     #"Ix Endstop Ext PX"
   //   A     #"Ix T1 Ret PX"
   //   A     #"Ix T2 Ext PX"
   //  R     #ClearPart."Reset Cyls for Idle"
   /////////////////  S     #Step.Idle

   ////////////////////////////////////////////////////////////////////////
   //end
END_REGION

REGION Network 7: Alarms
   // Because the HMI Alarms only works with INT data type, must set the individual address of the Data Block created: Alarms_DB
   //ESTOP
         A     #"ESTOP Pressed";
         =     %DB11.DBX0.0;

   //Doors
         AN    #"Ix Doors are Closed";
         =     %DB11.DBX0.1;

   //No Parts Timeout
         A     #No_Parts_Error;
         S     %DB11.DBX0.2;

   //bin is full
         A     "Bin_Count".Q;
         =     %DB11.DBX0.3;
END_REGION

REGION Network 8: Cylinder Jams
   // Cylinder Jam Logic for each ext and retract signal. 
   // Each one is 2 seconds and can be adjusted
   //blink Overhead lights when jammed
         A     #Cyl_Jam;
         AN    "Overhead_Blink".Q;
         =     #"Enable Overhead Blink";

         CALL  TON , "Overhead_Blink"
         ( IN := #"Enable Overhead Blink",
           PT := T#1s,
           Q  := ,
           ET :=
         );


   //------------------------------------------------------------
   //prestop
         A     #Auto."Prestop Cyl Ext";
         O     #Manual."Prestop Cyl Ext";
         O     #ClearPart."Extend Prestop";
         AN    #"Ix Prestop Ext PX";
         AN    #Pause;
         =     #Start_PreExt_Jam;

         CALL  TON, "Prestop_Ext_Jam_timer"
         ( IN := #Start_PreExt_Jam,
           PT := T#2s,
           Q  := ,
           ET :=
         );


         A     #Auto."Prestop Cyl Ret";
         O     #Manual."Prestop Cyl Ret";
         AN    #"Ix Prestop Ret PX";
         AN    #Pause;
         =     #Start_PreRet_Jam;

         CALL  TON , "Prestop_Ret_Jam_timer"
         ( IN := #Start_PreRet_Jam,
           PT := T#2s,
           Q  := ,
           ET :=
         );



   //------------------------------------------------------------
   //endstop
         A     #Auto."Endstop Cyl Ext";
         O     #Manual."Endstop Cyl Ext";
         AN    #"Ix Endstop Ext PX";
         AN    #Pause;
         =     #Start_EndExt_Jam;

         CALL  TON , "Endstop_Ext_Jam_timer"
         ( IN := #Start_EndExt_Jam,
           PT := T#2s,
           Q  := ,
           ET :=
         );


         A     #Auto."Endstop Cyl Ret";
         O     #Manual."Endstop Cyl Ret";
         O     #ClearPart."Retract Endstop";
         AN    #"Ix Endstop Ret PX";
         AN    #Pause;
         =     #Start_EndRet_Jam;

         CALL  TON , "Endstop_Ret_Jam_timer"
         ( IN := #Start_EndRet_Jam,
           PT := T#2s,
           Q  := ,
           ET :=
         );


   //------------------------------------------------------------
   //gripper

         A     #Auto."Gripper Cyl Ext";
         O     #Manual."Gripper Cyl Ext";
         O     #ClearPart."Extend Gripper";
         AN    #"Ix Gripper Ext PX";
         AN    #Pause;
         =     #Start_GrpExt_Jam;

         CALL  TON , "Gripper_Ext_Jam_timer"
         ( IN := #Start_GrpExt_Jam,
           PT := T#2s,
           Q  := ,
           ET :=
         );


         A     #Auto."Gripper Cyl Ret";
         O     #Manual."Gripper Cyl Ret";
         AN    #"Ix Gripper Ret PX";
         AN    #Pause;
         =     #Start_GrpRet_Jam;

         CALL  TON , "Gripper_Ret_Jam_timer"
         ( IN := #Start_GrpRet_Jam,
           PT := T#2s,
           Q  := ,
           ET :=
         );

   //------------------------------------------------------------
   //lat

         A     #Auto."Lat Cyl Ext";
         O     #Manual."Lat Cyl Ext";
         AN    #"Ix Lat Ext PX";
         AN    #Pause;
         =     #Start_LatExt_Jam;

         CALL  TON , "Lat_Ext_Jam_timer"
         ( IN := #Start_LatExt_Jam,
           PT := T#2s,
           Q  := ,
           ET :=
         );


         A     #Auto."Lat Cyl Ret";
         O     #Manual."Lat Cyl Ret";
         O     #ClearPart."Retract Lateral";
         AN    #"Ix Lat Ret PX";
         AN    #Pause;
         =     #Start_LatRet_Jam;

         CALL  TON , "Lat_Ret_Jam_timer"
         ( IN := #Start_LatRet_Jam,
           PT := T#2s,
           Q  := ,
           ET :=
         );


   //------------------------------------------------------------
   //clamp


         A     #Auto."Clamp Cyl Ext";
         O     #Manual."Clamp Cyl Ext";
         AN    #"Ix Left Clamp Ext PX";
         AN    #Pause;
         =     #Start_ClmpExt_Jam;

         CALL  TON , "Clamp_Ext_Jam_timer"
         ( IN := #Start_ClmpExt_Jam,
           PT := T#2s,
           Q  := ,
           ET :=
         );


         A     #Auto."Clamp Cyl Ret";
         O     #Manual."Clamp Cyl Ret";
         O     #ClearPart."Retract Clamp";
         AN    #"Ix Left Clamp Ret PX";
         AN    #Pause;
         =     #Start_ClmpRet_Jam;

         CALL  TON , "Clamp_Ret_Jam_timer"
         ( IN := #Start_ClmpRet_Jam,
           PT := T#2s,
           Q  := ,
           ET :=
         );

   //------------------------------------------------------------
   //shears

         A     #Auto."Shear Cyl Ext";
         O     #Manual."Shear Cyl Ext";
         AN    #"Ix Left Shear Ext PX";
         AN    #Pause;
         =     #Start_ShrExt_Jam;

         CALL  TON , "Shear_Ext_Jam_timer"
         ( IN := #Start_ShrExt_Jam,
           PT := T#2s,
           Q  := ,
           ET :=
         );


         A     #Auto."Shear Cyl Ret";
         O     #Manual."Shear Cyl Ret";
         O     #ClearPart."Retract Shears";
         AN    #"Ix Left Shear Ret PX";
         AN    #Pause;
         =     #Start_ShrRet_Jam;

         CALL  TON, "Shear_Ret_Jam_timer"
         ( IN := #Start_ShrRet_Jam,
           PT := T#2s,
           Q  := ,
           ET :=
         );

   //------------------------------------------------------------
   //punch

         A     #Auto."Punch Cyl Ext";
         O     #Manual."Punch Cyl Ext";
         AN    #"Ix Punch Ext PX";
         AN    #Pause;
         =     #Start_PunExt_Jam;

         CALL  TON, "Punch_Ext_Jam_timer"
         ( IN := #Start_PunExt_Jam,
           PT := T#2s,
           Q  := ,
           ET :=
         );


         A     #Auto."Punch Cyl Ret";
         O     #Manual."Punch Cyl Ret";
         O     #ClearPart."Retract Punch";
         AN    #"Ix Punch Ret PX";
         AN    #Pause;
         =     #Start_PunRet_Jam;

         CALL  TON, "Punch_Ret_Jam_timer"
         ( IN := #Start_PunRet_Jam,
           PT := T#2s,
           Q  := ,
           ET :=
         );


   //------------------------------------------------------------
   //T1
         A     #Auto."T1 Cyl Ext";
         O     #Manual."T1 Cyl Ext";
         AN    #"Ix T1 Ext PX";
         AN    #Pause;
         =     #Start_T1Ext_Jam;

         CALL  TON, "T1_Ext_Jam_timer"
         ( IN := #Start_T1Ext_Jam,
           PT := T#2s,
           Q  := ,
           ET :=
         );


         A     #Auto."T1 Cyl Ret";
         O     #Manual."T1 Cyl Ret";
         AN    #"Ix T1 Ret PX";
         AN    #Pause;
         =     #Start_T1Ret_Jam;

         CALL  TON, "T1_Ret_Jam_timer"
         ( IN := #Start_T1Ret_Jam,
           PT := T#2s,
           Q  := ,
           ET :=
         );


   //------------------------------------------------------------
   //T2
         A     #Auto."T2 Cyl Ext";
         O     #Manual."T2 Cyl Ext";
         AN    #"Ix T2 Ext PX";
         AN    #Pause;
         =     #Start_T2Ext_Jam;

         CALL  TON, "T2_Ext_Jam_timer"
         ( IN := #Start_T2Ext_Jam,
           PT := T#2s,
           Q  := ,
           ET :=
         );


         A     #Auto."T2 Cyl Ret";
         O     #Manual."T2 Cyl Ret";
         AN    #"Ix T2 Ret PX";
         AN    #Pause;
         =     #Start_T2Ret_Jam;

         CALL  TON, "T2_Ret_Jam_timer"
         ( IN := #Start_T2Ret_Jam,
           PT := T#2s,
           Q  := ,
           ET :=
         );



   //------------------------------------------------------------
   //Prompt an alarm for general cyl alarm
         A     "Prestop_Ext_Jam_timer".Q;
         O     "Prestop_Ret_Jam_timer".Q;

         O     "Endstop_Ext_Jam_timer".Q;
         O     "Endstop_Ret_Jam_timer".Q;

         O     "Gripper_Ext_Jam_timer".Q;
         O     "Gripper_Ret_Jam_timer".Q;

         O     "Lat_Ext_Jam_timer".Q;
         O     "Lat_Ret_Jam_timer".Q;

         O     "Clamp_Ext_Jam_timer".Q;
         O     "Clamp_Ret_Jam_timer".Q;

         O     "Shear_Ext_Jam_timer".Q;
         O     "Shear_Ret_Jam_timer".Q;

         O     "Punch_Ext_Jam_timer".Q;
         O     "Punch_Ret_Jam_timer".Q;

         O     "T1_Ext_Jam_timer".Q;
         O     "T1_Ret_Jam_timer".Q;

         O     "T2_Ext_Jam_timer".Q;
         O     "T2_Ret_Jam_timer".Q;

         =     #Cyl_Jam;
         S     %DB11.DBX0.4;

   //------------------------------------------------------------
   //individual cylinder alarms
         A     "Prestop_Ext_Jam_timer".Q;
         O     "Prestop_Ret_Jam_timer".Q;
         S     %DB11.DBX0.5;

         A     "Endstop_Ext_Jam_timer".Q;
         O     "Endstop_Ret_Jam_timer".Q;
         S     %DB11.DBX0.6;

         A     "Gripper_Ext_Jam_timer".Q;
         O     "Gripper_Ret_Jam_timer".Q;
         S     %DB11.DBX0.7;

         A     "Lat_Ext_Jam_timer".Q;
         O     "Lat_Ret_Jam_timer".Q;
         S     %DB11.DBX1.0;

         A     "Clamp_Ext_Jam_timer".Q;
         O     "Clamp_Ret_Jam_timer".Q;
         S     %DB11.DBX1.1;

         A     "Shear_Ext_Jam_timer".Q;
         O     "Shear_Ret_Jam_timer".Q;
         S     %DB11.DBX1.2;

         A     "Punch_Ext_Jam_timer".Q;
         O     "Punch_Ret_Jam_timer".Q;
         S     %DB11.DBX1.3;

         A     "T1_Ext_Jam_timer".Q;
         O     "T1_Ret_Jam_timer".Q;
         S     %DB11.DBX1.4;

         A     "T2_Ext_Jam_timer".Q;
         O     "T2_Ret_Jam_timer".Q;
         S     %DB11.DBX1.5;
END_REGION
END_FUNCTION_BLOCK

FUNCTION "FC_WintonWasher" : Void   // FC1, FBD
{ S7_Optimized_Access := 'FALSE' }
VERSION : 0.1
BEGIN

REGION Network 1
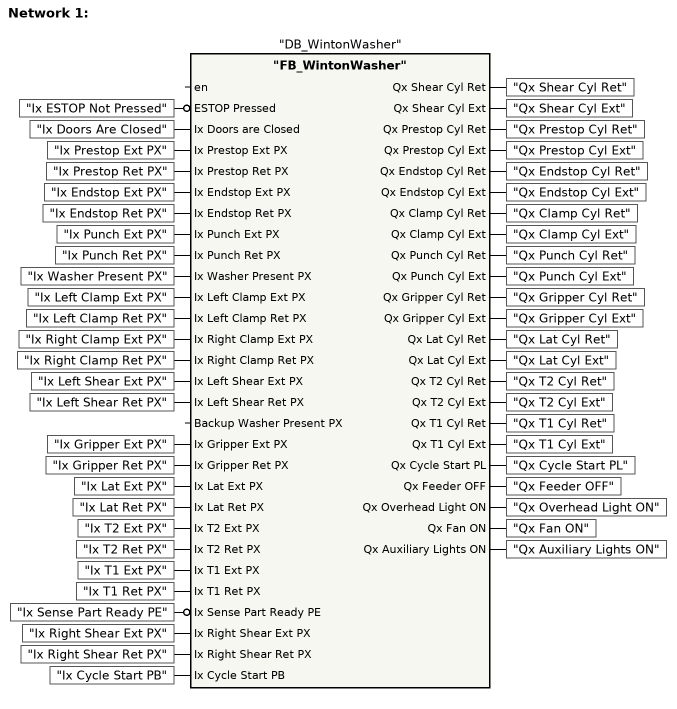
   "DB_WintonWasher"("ESTOP Pressed" := NOT "Ix ESTOP Not Pressed",   // "FB_WintonWasher"
                     "Ix Doors are Closed" := "Ix Doors Are Closed",
                     "Ix Prestop Ext PX" := "Ix Prestop Ext PX",
                     "Ix Prestop Ret PX" := "Ix Prestop Ret PX",
                     "Ix Endstop Ext PX" := "Ix Endstop Ext PX",
                     "Ix Endstop Ret PX" := "Ix Endstop Ret PX",
                     "Ix Punch Ext PX" := "Ix Punch Ext PX",
                     "Ix Punch Ret PX" := "Ix Punch Ret PX",
                     "Ix Washer Present PX" := "Ix Washer Present PX",
                     "Ix Left Clamp Ext PX" := "Ix Left Clamp Ext PX",
                     "Ix Left Clamp Ret PX" := "Ix Left Clamp Ret PX",
                     "Ix Right Clamp Ext PX" := "Ix Right Clamp Ext PX",
                     "Ix Right Clamp Ret PX" := "Ix Right Clamp Ret PX",
                     "Ix Left Shear Ext PX" := "Ix Left Shear Ext PX",
                     "Ix Left Shear Ret PX" := "Ix Left Shear Ret PX",
                     "Ix Gripper Ext PX" := "Ix Gripper Ext PX",
                     "Ix Gripper Ret PX" := "Ix Gripper Ret PX",
                     "Ix Lat Ext PX" := "Ix Lat Ext PX",
                     "Ix Lat Ret PX" := "Ix Lat Ret PX",
                     "Ix T2 Ext PX" := "Ix T2 Ext PX",
                     "Ix T2 Ret PX" := "Ix T2 Ret PX",
                     "Ix T1 Ext PX" := "Ix T1 Ext PX",
                     "Ix T1 Ret PX" := "Ix T1 Ret PX",
                     "Ix Sense Part Ready PE" := NOT "Ix Sense Part Ready PE",
                     "Ix Right Shear Ext PX" := "Ix Right Shear Ext PX",
                     "Ix Right Shear Ret PX" := "Ix Right Shear Ret PX",
                     "Ix Cycle Start PB" := "Ix Cycle Start PB",
                     "Qx Shear Cyl Ret" => "Qx Shear Cyl Ret",
                     "Qx Shear Cyl Ext" => "Qx Shear Cyl Ext",
                     "Qx Prestop Cyl Ret" => "Qx Prestop Cyl Ret",
                     "Qx Prestop Cyl Ext" => "Qx Prestop Cyl Ext",
                     "Qx Endstop Cyl Ret" => "Qx Endstop Cyl Ret",
                     "Qx Endstop Cyl Ext" => "Qx Endstop Cyl Ext",
                     "Qx Clamp Cyl Ret" => "Qx Clamp Cyl Ret",
                     "Qx Clamp Cyl Ext" => "Qx Clamp Cyl Ext",
                     "Qx Punch Cyl Ret" => "Qx Punch Cyl Ret",
                     "Qx Punch Cyl Ext" => "Qx Punch Cyl Ext",
                     "Qx Gripper Cyl Ret" => "Qx Gripper Cyl Ret",
                     "Qx Gripper Cyl Ext" => "Qx Gripper Cyl Ext",
                     "Qx Lat Cyl Ret" => "Qx Lat Cyl Ret",
                     "Qx Lat Cyl Ext" => "Qx Lat Cyl Ext",
                     "Qx T2 Cyl Ret" => "Qx T2 Cyl Ret",
                     "Qx T2 Cyl Ext" => "Qx T2 Cyl Ext",
                     "Qx T1 Cyl Ret" => "Qx T1 Cyl Ret",
                     "Qx T1 Cyl Ext" => "Qx T1 Cyl Ext",
                     "Qx Cycle Start PL" => "Qx Cycle Start PL",
                     "Qx Feeder OFF" => "Qx Feeder OFF",
                     "Qx Overhead Light ON" => "Qx Overhead Light ON",
                     "Qx Fan ON" => "Qx Fan ON",
                     "Qx Auxiliary Lights ON" => "Qx Auxiliary Lights ON");
END_REGION
END_FUNCTION

ORGANIZATION_BLOCK "Main"   // OB1, STL
TITLE = "Main Program Sweep (Cycle)"
{ S7_Optimized_Access := 'FALSE' }
VERSION : 0.1
   VAR_TEMP
      OB1_EV_CLASS : Byte;   // Bits 0-3 = 1 (Coming event), Bits 4-7 = 1 (Event class 1)
      OB1_SCAN_1 : Byte;   // 1 (Cold restart scan 1 of OB 1), 3 (Scan 2-n of OB 1)
      OB1_PRIORITY : Byte;   // Priority of OB Execution
      OB1_OB_NUMBR : Byte;   // 1 (Organization block 1, OB1)
      OB1_RESERVED_1 : Byte;   // Reserved for system
      OB1_RESERVED_2 : Byte;   // Reserved for system
      OB1_PREV_CYCLE : Int;   // Cycle time of previous OB1 scan (milliseconds)
      OB1_MIN_CYCLE : Int;   // Minimum cycle time of OB1 (milliseconds)
      OB1_MAX_CYCLE : Int;   // Maximum cycle time of OB1 (milliseconds)
      OB1_DATE_TIME : Date_And_Time;   // Date and time OB1 started
   END_VAR
BEGIN

REGION Network 1
         CALL  "FC_WintonWasher";
END_REGION
END_ORGANIZATION_BLOCK

(* ===== HMI "HMI_RT_1" =====
system functions are stored by id; their names below are inferred from use
connection "HMI_Connection": ETHERNET, SIMATIC S7 300/400 MPI

HMI tags "HMI Tag Table"
   "HMI_MasterReset" : Bool = PLC HMI_DB.MasterReset AT %DB7.DBX0.0, 1 s
   "HMI Prestop Ext" : Bool = PLC HMI_DB."Prestop Ext" AT %DB7.DBX0.7, 1 s
   "HMI Prestop Ret" : Bool = PLC HMI_DB."Prestop Ret" AT %DB7.DBX1.0, 1 s
   "HMI Endstop Ext" : Bool = PLC HMI_DB."Endstop Ext" AT %DB7.DBX1.1, 1 s
   "HMI Endstop Ret" : Bool = PLC HMI_DB."Endstop Ret" AT %DB7.DBX1.2, 1 s
   "HMI Lat Ext" : Bool = PLC HMI_DB."Lat Ext" AT %DB7.DBX1.7, 1 s
   "HMI Lat Ret" : Bool = PLC HMI_DB."Lat Ret" AT %DB7.DBX2.0, 1 s
   "HMI Punch Ret" : Bool = PLC HMI_DB."Punch Ret" AT %DB7.DBX0.4, 1 s
   "HMI Gripper Ext" : Bool = PLC HMI_DB."Gripper Ext" AT %DB7.DBX1.5, 1 s
   "HMI Gripper Ret" : Bool = PLC HMI_DB."Gripper Ret" AT %DB7.DBX1.6, 1 s
   "HMI T1 Ext" : Bool = PLC HMI_DB."T1 Ext" AT %DB7.DBX2.1, 1 s
   "HMI T1 Ret" : Bool = PLC HMI_DB."T1 Ret" AT %DB7.DBX2.2, 1 s
   "HMI T2 Ext" : Bool = PLC HMI_DB."T2 Ext" AT %DB7.DBX2.3, 1 s
   "HMI T2 Ret" : Bool = PLC HMI_DB."T2 Ret" AT %DB7.DBX2.4, 1 s
   "HMI Shear Ext" : Bool = PLC HMI_DB."Shear Ext" AT %DB7.DBX0.5, 1 s
   "HMI Shear Ret" : Bool = PLC HMI_DB."Shear Ret" AT %DB7.DBX0.6, 1 s
   "HMI Clamp Ext" : Bool = PLC HMI_DB."Clamp Ext" AT %DB7.DBX1.3, 1 s
   "HMI Clamp Ret" : Bool = PLC HMI_DB."Clamp Ret" AT %DB7.DBX1.4, 1 s
   "HMI Auto ON" : Bool = PLC HMI_DB."Auto On" AT %DB7.DBX0.2, 1 s
   "Ix Prestop Ext PX" : Bool = PLC "Ix Prestop Ext PX" AT %I10.2, 1 s
   "Ix Prestop Ret PX" : Bool = PLC "Ix Prestop Ret PX" AT %I10.3, 1 s
   "Ix T1 Ext PX" : Bool = PLC "Ix T1 Ext PX" AT %I12.6, 1 s
   "Ix T1 Ret PX" : Bool = PLC "Ix T1 Ret PX" AT %I12.7, 1 s
   "Ix T2 Ext PX" : Bool = PLC "Ix T2 Ext PX" AT %I12.4, 1 s
   "Ix T2 Ret PX" : Bool = PLC "Ix T2 Ret PX" AT %I12.5, 1 s
   "Ix Lat Ext PX" : Bool = PLC "Ix Lat Ext PX" AT %I12.2, 1 s
   "Ix Lat Ret PX" : Bool = PLC "Ix Lat Ret PX" AT %I12.3, 1 s
   "Ix Doors Are Closed" : Bool = PLC "Ix Doors Are Closed" AT %I1.2, 1 s
   "Ix Punch Ext PX" : Bool = PLC "Ix Punch Ext PX" AT %I10.6, 1 s
   "Ix Punch Ret PX" : Bool = PLC "Ix Punch Ret PX" AT %I10.7, 1 s
   "Ix Left Clamp Ext PX" : Bool = PLC "Ix Left Clamp Ext PX" AT %I11.2, 1 s
   "Ix Left Clamp Ret PX" : Bool = PLC "Ix Left Clamp Ret PX" AT %I11.3, 1 s
   "Ix Right Clamp Ext PX" : Bool = PLC "Ix Right Clamp Ext PX" AT %I11.4, 1 s
   "Ix Right Clamp Ret PX" : Bool = PLC "Ix Right Clamp Ret PX" AT %I11.5, 1 s
   "Ix Right Shear Ext PX" : Bool = PLC "Ix Right Shear Ext PX" AT %I13.6, 1 s
   "Ix Right Shear Ret PX" : Bool = PLC "Ix Right Shear Ret PX" AT %I13.7, 1 s
   "Ix ESTOP Not Pressed" : Bool = PLC "Ix ESTOP Not Pressed" AT %I1.1, 1 s
   "Ix Sense Part Ready PE" : Bool = PLC "Ix Sense Part Ready PE" AT %I13.4, 1 s
   "Ix Washer Present PX" : Bool = PLC "Ix Washer Present PX" AT %I11.0, 1 s
   "Ix Endstop Ext PX" : Bool = PLC "Ix Endstop Ext PX" AT %I10.4, 1 s
   "Ix Endstop Ret PX" : Bool = PLC "Ix Endstop Ret PX" AT %I10.5, 1 s
   "Ix Gripper Ext PX" : Bool = PLC "Ix Gripper Ext PX" AT %I12.0, 1 s
   "Ix Gripper Ret PX" : Bool = PLC "Ix Gripper Ret PX" AT %I12.1, 1 s
   "Ix Cycle Start PB" : Bool = PLC "Ix Cycle Start PB" AT %I1.0, 1 s
   "HMI Punch Ext" : Bool = PLC HMI_DB."Punch Ext" AT %DB7.DBX0.3, 1 s
   "HMI Aux Lights" : Bool = PLC HMI_DB."Auxiliary Lights" AT %DB7.DBX2.7, 1 s
   "HMI Overhead Lights" : Bool = PLC HMI_DB."Overhead Lights" AT %DB7.DBX2.6, 1 s
   "Ix Part Present" : Bool = PLC "Ix Sense Part Ready PE" AT %I13.4, 1 s
   "HMI_Pause" : Bool = PLC HMI_DB.Pause AT %DB7.DBX0.1, 1 s
   "Ix Left Shear Ret PX" : Bool = PLC "Ix Left Shear Ret PX" AT %I11.7, 1 s
   "Ix Left Shear Ext PX" : Bool = PLC "Ix Left Shear Ext PX" AT %I11.6, 1 s
   "Qx Vibrate OFF" : Bool = PLC "Qx Feeder OFF" AT %Q5.1, 1 s
   "HMI Vibrate" : Bool = PLC HMI_DB.Vibrate AT %DB7.DBX2.5, 1 s
   "Bin_Count" : Int = PLC HMI_DB.Bin_Count AT %DB7.DBW4, 1 s
   "HMI Fan" : Bool = PLC HMI_DB.Fan AT %DB7.DBX3.0, 1 s
   "Reset_Bin_Count" : Bool = PLC HMI_DB.Reset_Bin_Count AT %DB7.DBX6.0, 1 s
   "Cycle_Count" : Int = PLC HMI_DB.Cycle_Count AT %DB7.DBW8, 1 s
   "Alarms" : Word = PLC Alarms_DB.Alarms AT %DB11.DBW0, 1 s

discrete alarms
   1: 'ESTOP PRESSED: Release When Ready For Idle', class Warnings, trigger "Alarms" bit 8
   2: 'DOORS OPEN: Close Doors to Continue', class Warnings, trigger "Alarms" bit 9
   3: 'FEEDER TIMEOUT: Clear Pop-Up Button, Load Parts and Press Cycle Start to Continue', class Warnings, trigger "Alarms" bit 10
   4: 'BIN FULL: Empty Bin and Reset Bin Count to Continue', class Warnings, trigger "Alarms" bit 11
   5: 'Cyl Jam. Master Reset in Auto to attempt to clear part. Manually clear otherwise', class Warnings, trigger "Alarms" bit 12
   6: 'Prestop is Jammed', class Warnings, trigger "Alarms" bit 13
   7: 'Endstop is Jammed', class Warnings, trigger "Alarms" bit 14
   8: 'Gripper is Jammed', class Warnings, trigger "Alarms" bit 15
   9: 'Lateral is Jammed', class Warnings, trigger "Alarms" bit 0
   10: 'Clamp is Jammed', class Warnings, trigger "Alarms" bit 1
   11: 'Shear is Jammed', class Warnings, trigger "Alarms" bit 2
   12: 'Punch is Jammed', class Warnings, trigger "Alarms" bit 3
   13: 'Trap Door 1 is Jammed', class Warnings, trigger "Alarms" bit 4
   14: 'Trap Door 2 is Jammed', class Warnings, trigger "Alarms" bit 5

screen "Main Screen" 800x420, template "Template_1"
   Button "Button_2" at 274,187 size 236x70; TextOff 'Pause'
      Appearance <- "HMI_Pause"
      on Press: InvertBit("HMI_Pause")
   TextField "Text field_1" at 288,172 size 16x23; Text 'Text'
   Button "Button_8" at 191,264 size 184x98; TextOff 'Manual Cyl Control'
      on Press: ActivateScreen("Manual_Cyls", 0)
   Button "Button_7" at 6,264 size 168x98; TextOff 'Input Monitor'
      on Press: ActivateScreen("Input Monitor", 0)
   TextField "Text field_2" at 289,4 size 212x43; Text 'Main Screen'
   Button "Button_9" at 638,264 size 157x98; TextOff 'Alarms'
      on Press: ActivateScreen("Alarm Info", 0)
   Button "Auto Button" at 275,57 size 233x124; TextOff 'Auto Run'
      Appearance <- "HMI Auto ON"
      ProcessValue <- "HMI Auto ON"
      on Press: InvertBit("HMI Auto ON")
   Button "Button_1" at 392,264 size 230x98; TextOff 'Manual Peripheral Control'
      on Press: ActivateScreen("Manual_Etc", 0)
   TextField "Text field_3" at 625,62 size 104x25; Text 'Bin Count'
   Button "Button_3" at 566,179 size 220x68; TextOff 'Reset Bin Count'
      on Press: function_b14e0dd5("Reset_Bin_Count", 0)
   Bar "Bar_1" at 558,89 size 233x80; MinimumValue 0; MaximumValue 135
      ProcessValue <- "Bin_Count"
   Button "Button_5" at 4,57 size 200x114; TextOff 'Master Reset'
      on Press: function_b14e0dd5("HMI_MasterReset", 0); function_a9b64e44("Alarms", 12); function_a9b64e44("Alarms", 13); function_a9b64e44("Alarms", 14); function_a9b64e44("Alarms", 0); function_a9b64e44("Alarms", 1); function_a9b64e44("Alarms", 2); function_a9b64e44("Alarms", 3); function_a9b64e44("Alarms", 4); function_a9b64e44("Alarms", 5)
      Appearance <- "HMI_MasterReset"
   Rectangle "Rectangle_3" at 158,367 size 140x49
      Appearance <- "Alarms"
      Visibility <- "Alarms"
   TextField "Text field_4" at 162,379 size 141x23; Text 'ESTOP Pressed'
      Visibility <- "Alarms"
   Rectangle "Rectangle_4" at 302,367 size 129x49
      Appearance <- "Alarms"
      Visibility <- "Alarms"
   TextField "Text field_5" at 306,379 size 112x23; Text 'DOOR OPEN'
      Visibility <- "Alarms"
   Rectangle "Rectangle_6" at 436,367 size 115x49
      Appearance <- "Alarms"
      Visibility <- "Alarms"
   TextField "Text field_7" at 443,379 size 87x23; Text 'BIN FULL'
      Visibility <- "Alarms"
   TextField "Text field_6" at 4,231 size 93x29; Text 'Screens'
   Button "Button_4" at 7,179 size 230x56; TextOff 'CYL JAM: See Alarms'
      on Click: function_a9b64e44("Alarms", 10)
      Visibility <- "Alarms"
      Appearance <- "Alarms"
   Button "Button_6" at 255,119 size 283x108; TextOff 'FEEDER TIMEOUT: Load Parts'
      on Click: function_a9b64e44("Alarms", 10)
      Visibility <- "Alarms"

screen "Manual_Cyls" 800x420
   Button "Button_1" at 709,343 size 87x75; TextOff 'Text'; PictureOff "Home"
      on Click: ActivateScreen("Main Screen", 0)
   TextField "Text field_1" at 215,8 size 380x37; Text 'Manual Control: Cylinders'
   TextField "Text field_3" at 7,78 size 93x29; Text 'Prestop'
   Button "Button_3" at 113,67 size 110x56; TextOff 'RET'
      Appearance <- "Ix Prestop Ret PX"
      on Press: function_b14e0dd5("HMI Prestop Ret", 0)
   Button "Button_11" at 262,67 size 110x56; TextOff 'EXT'
      Appearance <- "Ix Prestop Ext PX"
      on Press: function_b14e0dd5("HMI Prestop Ext", 0)
   TextField "Text field_2" at 7,152 size 97x29; Text 'Endstop'
   Button "Button_2" at 111,139 size 110x57; TextOff 'RET'
      on Press: function_b14e0dd5("HMI Endstop Ret", 0)
      Appearance <- "Ix Endstop Ret PX"
   Button "Button_4" at 262,139 size 110x57; TextOff 'EXT'
      Appearance <- "Ix Endstop Ext PX"
      on Press: function_b14e0dd5("HMI Endstop Ext", 0)
   TextField "Text field_6" at 8,295 size 86x29; Text 'Lateral'
   Button "Button_5" at 108,283 size 110x55; TextOff 'RET'
      on Press: function_b14e0dd5("HMI Lat Ret", 0)
      Appearance <- "Ix Lat Ret PX"
   Button "Button_6" at 262,283 size 110x55; TextOff 'EXT'
      Appearance <- "Ix Lat Ext PX"
      on Press: function_b14e0dd5("HMI Lat Ext", 0)
   TextField "Text field_7" at 8,224 size 90x29; Text 'Gripper'
   Button "Button_7" at 109,212 size 110x57; TextOff 'RET'
      on Press: function_b14e0dd5("HMI Gripper Ret", 0)
      Appearance <- "Ix Gripper Ret PX"
   Button "Button_8" at 263,212 size 110x57; TextOff 'EXT'
      Appearance <- "Ix Gripper Ext PX"
      on Press: function_b14e0dd5("HMI Gripper Ext", 0)
   TextField "Text field_10" at 390,80 size 76x29; Text 'Clamp'
   Button "Button_9" at 500,67 size 110x56; TextOff 'RET'
      on Press: function_b14e0dd5("HMI Clamp Ret", 0)
      Appearance <- "Ix Right Clamp Ret PX"
   Button "Button_12" at 650,67 size 110x56; TextOff 'EXT'
      Appearance <- "Ix Right Clamp Ext PX"
      on Press: function_b14e0dd5("HMI Clamp Ext", 0)
   TextField "Text field_11" at 391,153 size 63x25; Text 'Punch'
   Button "Button_13" at 500,140 size 110x56; TextOff 'RET'
      on Press: function_b14e0dd5("HMI Punch Ret", 0)
      Appearance <- "Ix Punch Ret PX"
   Button "Button_14" at 650,140 size 110x56; TextOff 'EXT'
      Appearance <- "Ix Punch Ext PX"
      on Press: function_b14e0dd5("HMI Punch Ext", 0)
   TextField "Text field_13" at 391,227 size 117x25; Text 'Trap Door 1'
   Button "Button_15" at 500,211 size 110x57; TextOff 'RET'
      on Press: function_b14e0dd5("HMI T1 Ret", 0)
      Appearance <- "Ix T1 Ret PX"
   Button "Button_16" at 650,211 size 110x57; TextOff 'EXT'
      Appearance <- "Ix T1 Ext PX"
      on Press: function_b14e0dd5("HMI T1 Ext", 0)
   TextField "Text field_14" at 393,298 size 117x25; Text 'Trap Door 2'
   Button "Button_17" at 500,282 size 110x56; TextOff 'RET'
      on Press: function_b14e0dd5("HMI T2 Ret", 0)
      Appearance <- "Ix T2 Ret PX"
   Button "Button_18" at 650,282 size 110x56; TextOff 'EXT'
      Appearance <- "Ix T2 Ext PX"
      on Press: function_b14e0dd5("HMI T2 Ext", 0)
   TextField "Text field_15" at 202,343 size 82x29; Text 'Shears'
   TextField "Text field_5" at 189,388 size 61x22; Text 'Right:'
   TextField "Text field_8" at 191,370 size 50x22; Text 'Left:'
   Button "Button_22" at 326,347 size 102x69; TextOff 'RET'
      on Press: function_b14e0dd5("HMI Shear Ret", 0)
      Appearance <- "Ix Left Shear Ret PX"
   Button "Button_19" at 486,347 size 102x69; TextOff 'EXT'
      on Press: function_b14e0dd5("HMI Shear Ret", 0)
      Appearance <- "Ix Left Shear Ext PX"
   Circle "Circle_18" at 295,364 size 25x25
      Appearance <- "Ix Left Shear Ret PX"
   Circle "Circle_1" at 295,389 size 25x25
      Appearance <- "Ix Right Shear Ret PX"
   Circle "Circle_2" at 455,363 size 25x25
      Appearance <- "Ix Left Shear Ext PX"
   Circle "Circle_3" at 455,388 size 25x25
      Appearance <- "Ix Right Shear Ext PX"

screen "Alarm Info" 800x420
   Button "Button_1" at 702,337 size 87x75; TextOff 'Text'; PictureOff "Home"
      on Click: ActivateScreen("Main Screen", 0)
   AlarmView "Alarm view_1" at 8,40 size 683x372
   TextField "Text field_1" at 8,1 size 200x34; Text 'Alarm History'

screen "Input Monitor" 800x420
   Button "Button_1" at 724,368 size 66x50; TextOff 'Text'; PictureOff "Home"
      on Click: ActivateScreen("Main Screen", 0)
   TextField "Text field_28" at 51,105 size 194x25; Text 'Prestop is Retracted'
   TextField "Text field_32" at 306,104 size 178x25; Text 'Punch is Retracted'
   TextField "Text field_50" at 51,299 size 174x25; Text 'Cycle Start Button'
   TextField "Text field_52" at 494,379 size 194x29; Text 'Doors Are Closed'
   TextField "Text field_27" at 51,71 size 189x25; Text 'Prestop is Extended'
   TextField "Text field_31" at 308,69 size 173x25; Text 'Punch is Extended'
   TextField "Text field_33" at 51,379 size 180x25; Text 'Washer Present PX'
   TextField "Text field_47" at 50,338 size 137x25; Text 'Part Ready PE'
   TextField "Text field_1" at 305,7 size 207x37; Text 'Input Monitor'
   Circle "Circle_18" at 9,69 size 29x29
      Appearance <- "Ix Prestop Ext PX"
   Circle "Circle_9" at 9,102 size 29x29
      Appearance <- "Ix Prestop Ret PX"
   Circle "Circle_1" at 270,67 size 29x29
      Appearance <- "Ix Punch Ext PX"
   Circle "Circle_2" at 269,100 size 29x29
      Appearance <- "Ix Punch Ret PX"
   TextField "Text field_4" at 591,103 size 147x25; Text 'T1 is Retracted'
   TextField "Text field_5" at 592,69 size 142x25; Text 'T1 is Extended'
   Circle "Circle_19" at 544,67 size 29x29
      Appearance <- "Ix Prestop Ext PX"
   Circle "Circle_27" at 544,100 size 29x29
      Appearance <- "Ix Prestop Ext PX"
   TextField "Text field_3" at 51,181 size 196x25; Text 'Endstop is Retracted'
   TextField "Text field_6" at 306,180 size 192x25; Text 'Gripper is Retracted'
   TextField "Text field_7" at 51,147 size 191x25; Text 'Endstop is Extended'
   TextField "Text field_8" at 308,145 size 187x25; Text 'Gripper is Extended'
   Circle "Circle_3" at 9,145 size 29x29
      Appearance <- "Ix Endstop Ext PX"
   Circle "Circle_4" at 9,178 size 29x29
      Appearance <- "Ix Endstop Ret PX"
   Circle "Circle_5" at 270,143 size 29x29
      Appearance <- "Ix Gripper Ext PX"
   Circle "Circle_6" at 269,176 size 29x29
      Appearance <- "Ix Gripper Ret PX"
   TextField "Text field_9" at 591,179 size 153x25; Text 'T2 is Retracted'
   TextField "Text field_10" at 592,145 size 142x25; Text 'T2 is Extended'
   Circle "Circle_10" at 544,143 size 29x29
      Appearance <- "Ix Prestop Ext PX"
   Circle "Circle_12" at 544,176 size 29x29
      Appearance <- "Ix Prestop Ext PX"
   TextField "Text field_11" at 52,256 size 189x25; Text 'Lateral is Retracted'
   TextField "Text field_12" at 306,254 size 224x25; Text 'Left Shear is Retracted'
   TextField "Text field_13" at 52,222 size 184x25; Text 'Lateral is Extended'
   TextField "Text field_14" at 307,222 size 213x25; Text 'Left Shear is Extended'
   Circle "Circle_13" at 10,220 size 29x29
      Appearance <- "Ix Lat Ext PX"
   Circle "Circle_14" at 10,253 size 29x29
      Appearance <- "Ix Lat Ret PX"
   Circle "Circle_17" at 270,218 size 29x29
      Appearance <- "Ix Left Shear Ext PX"
   Circle "Circle_20" at 270,251 size 29x29
      Appearance <- "Ix Left Shear Ret PX"
   TextField "Text field_17" at 566,255 size 231x25; Text 'Right Shear is Retracted'
   TextField "Text field_18" at 568,223 size 226x25; Text 'Right Shear is Extended'
   Circle "Circle_23" at 535,221 size 29x29
      Appearance <- "Ix Right Shear Ext PX"
   Circle "Circle_24" at 535,253 size 29x29
      Appearance <- "Ix Right Shear Ret PX"
   TextField "Text field_2" at 305,333 size 228x25; Text 'Left Clamp is Retracted'
   TextField "Text field_15" at 306,300 size 217x25; Text 'Left Clamp is Extended'
   TextField "Text field_16" at 565,332 size 235x25; Text 'Right Clamp is Retracted'
   TextField "Text field_19" at 566,300 size 230x25; Text 'Right Clamp is Extended'
   Circle "Circle_7" at 534,298 size 29x29
      Appearance <- "Ix Right Clamp Ext PX"
   Circle "Circle_8" at 535,330 size 29x29
      Appearance <- "Ix Right Clamp Ret PX"
   Circle "Circle_21" at 270,298 size 29x29
      Appearance <- "Ix Left Clamp Ext PX"
   Circle "Circle_22" at 270,330 size 29x29
      Appearance <- "Ix Left Clamp Ret PX"
   Circle "Circle_11" at 11,298 size 29x29
      Appearance <- "Ix Cycle Start PB"
   Circle "Circle_25" at 11,377 size 29x29
      Appearance <- "Ix Washer Present PX"
   Circle "Circle_26" at 11,336 size 29x29
      Appearance <- "Ix Sense Part Ready PE"
   TextField "Text field_20" at 312,379 size 103x29; Text 'Estop OK'
   Circle "Circle_15" at 264,372 size 41x41
      Appearance <- "Ix ESTOP Not Pressed"
   Circle "Circle_28" at 446,372 size 41x41
      Appearance <- "Ix Doors Are Closed"

Template "Template_1" 800x420
   Button "Exit" at 720,360 size 78x58; TextOff 'Exit'; PictureOff "ExitRuntime_TP700_Comfort_TR"; PictureOn "ExitRuntime_TP700_Comfort_TR"
      on Release: StopRuntime(0)
   Button "Template_Button" at 640,360 size 78x58; TextOff 'Text'
   Button "Template_Button_1" at 560,360 size 78x58; TextOff 'Text'
   Button "Template_Button_2" at 480,360 size 78x58; TextOff 'Text'
   Button "Template_Button_3" at 400,360 size 78x58; TextOff 'Text'
   Button "Template_Button_4" at 321,360 size 78x58; TextOff 'Text'
   Button "Template_Button_5" at 241,360 size 78x58; TextOff 'Text'
   Button "Template_Button_6" at 161,360 size 78x58; TextOff 'Text'
   Button "Alarms" at 81,360 size 78x58; TextOff 'Alarms'; PictureOff "AlarmDisplay_TP700_Comfort_TR"; PictureOn "AlarmDisplay_TP700_Comfort_TR"
      on Release: function_ef3f5d25("Alarm window_Unacknowledged", -1)
   Button "Start screen" at 1,360 size 78x58; TextOff 'Start screen'; PictureOff "NavigateHome_TP700_Comfort_TR"; PictureOn "NavigateHome_TP700_Comfort_TR"
      on Release: ActivateScreen("Main Screen", 0)

screen "Manual_Etc" 800x420
   TextField "Text field_1" at 40,82 size 150x27; Text 'Vibrating Rail'
   Button "Button_2" at 270,80 size 98x95; TextOff 'Toggle'
      on Press: InvertBit("HMI Vibrate")
   TextField "Text field_2" at 124,118 size 51x39; Text 'ON'
      Appearance <- "Qx Vibrate OFF"
   TextField "Text field_3" at 187,118 size 63x39; Text 'OFF'
      Appearance <- "Qx Vibrate OFF"
   TextField "Text field_4" at 218,8 size 384x37; Text 'Manual Peripheral Control'
   Button "Button_1" at 709,343 size 87x75; TextOff 'Text'; PictureOff "Home"
      on Click: ActivateScreen("Main Screen", 0)
   TextField "Text field_5" at 40,190 size 165x27; Text 'Overhead Light'
   Button "Button_3" at 270,188 size 98x95; TextOff 'Toggle'
      on Press: InvertBit("HMI Overhead Lights")
   TextField "Text field_6" at 124,226 size 51x39; Text 'ON'
      Appearance <- "HMI Overhead Lights"
   TextField "Text field_7" at 187,226 size 63x39; Text 'OFF'
      Appearance <- "HMI Overhead Lights"
   TextField "Text field_8" at 430,190 size 170x27; Text 'Auxiliary Lights'
   Button "Button_4" at 660,188 size 98x95; TextOff 'Toggle'
      on Press: InvertBit("HMI Aux Lights")
   TextField "Text field_9" at 514,226 size 51x39; Text 'ON'
      Appearance <- "HMI Aux Lights"
   TextField "Text field_10" at 577,226 size 63x39; Text 'OFF'
      Appearance <- "HMI Aux Lights"
   TextField "Text field_11" at 431,82 size 46x29; Text 'Fan'
   Button "Button_5" at 661,80 size 98x95; TextOff 'Toggle'
      on Press: InvertBit("HMI Fan")
   TextField "Text field_12" at 515,118 size 51x39; Text 'ON'
      Appearance <- "HMI Fan"
   TextField "Text field_13" at 578,118 size 63x39; Text 'OFF'
      Appearance <- "HMI Fan"
   IOField "I/O field_1" at 264,321 size 268x94; FormatPattern 99999
      ProcessValue <- "Cycle_Count"
   TextField "Text field_14" at 311,291 size 190x32; Text 'Parts Recycled'
*)